TYPE ST_INPUTS_Unit_RO_EDI:
STRUCT
	
	Mode:     		E_DeviceMode;
	Command:     	E_DeviceState;

END_STRUCT
END_TYPE

(* stored: Version 1.1.0.1, ProductVersion 3.1.4024.12
   DUT ST_INPUTS_Unit_RO_EDI: Id {d074f931-2cd0-4789-b5e1-e2e58df6cf7b} *)
